INTERFACE I_PwmLightTowerComponent EXTENDS I_LightTowerComponent

// Starts the pulse width modulation of the component.
METHOD Activate
VAR_INPUT
END_VAR
END_METHOD

// Stop the pulse width modulation of the component.
METHOD Deactivate
VAR_INPUT
END_VAR
END_METHOD

// Sets the interval of the PWM to desired value tInterval.
METHOD SetInterval : I_LightTowerComponent
VAR_INPUT
	tInterval	: TIME;
END_VAR
END_METHOD

END_INTERFACE

(* stored: Version 1.1.0.1, ProductVersion 3.1.4024.13
   Itf I_PwmLightTowerComponent: Id {9513e11e-a9b1-07cf-382b-49c95a4f2b7b}
   Method Activate: Id {a04d9040-272a-0b91-10e6-a5bdf954aff7}
   Method Deactivate: Id {0da7f011-c57a-0fca-1b8d-23f37beb95e2}
   Method SetInterval: Id {1eb69c19-1edc-0a86-02be-65d866bd735d} *)
